// TwinCAT 3 PLC project motor_test1
// ProgramVersion: 3.1.0.9
// libraries:
//   VisuElem3DPath, 3.5.4.0 (System)
//   VisuElemMeter, 3.5.4.0 (System)
//   VisuElems, 3.5.4.10 (System)
//   VisuElemsSpecialControls, 3.5.4.10 (System)
//   VisuElemsWinControls, 3.5.4.10 (System)
//   VisuElemTextEditor, 3.5.4.0 (System)
//   visuinputs, 3.5.4.0 (system)
//   VisuNativeControl, 3.5.4.0 (System)
//   Tc2_Standard, * (Beckhoff Automation GmbH)
//   Tc2_System, * (Beckhoff Automation GmbH)
//   Tc2_Utilities, * (Beckhoff Automation GmbH)
//   Tc3_Interfaces, * (Beckhoff Automation GmbH)
//   Tc3_Module, * (Beckhoff Automation GmbH)
//   VisuDialogs, * (System)
//   Tc2_MC2,3.3.8.0,Beckhoff Automation GmbH
//   Tc2_SerialCom,3.3.3.0,Beckhoff Automation GmbH
// project tree:
//   / FastTask.TcTTO, GlobalTextList.TcGTLO, PlcTask.TcTTO, Visualization Manager.TcVMO (not stored)
//   GVLs/ GVL.TcGVL
//   POUs/ allgemein.TcPOU, Background.TcPOU, BackgroundEL.TcPOU, MAIN.TcPOU, resetErrorHandling.TcPOU, SerialCom.TcPOU, visu.TcPOU, writeInArray.TcPOU (not stored)
//   VISUs/ ImageCollection.TcIPO (not stored), AutomaticMode.TcVIS, startView.TcVIS
// real-time tasks:
//   TASK PlcTask: cycle T#5ms, priority 20, ADS port 351
//   TASK FastTask: cycle T#1ms, priority 10, ADS port 350
// motion (NC):
//   TASK NC-Task 1 SAF: cycle T#2ms, priority 4, ADS port 501
//   TASK NC-Task 1 SVB: cycle T#10ms, priority 8, ADS port 511
//   AXIS Axis Y (id 1)
//     Dynamic: Acceleration=3000, Deceleration=3000, Jerk=500
//     Velo: RefSearch=10, RefSync=10, SlowManual=10, FastManual=100, Maximum=400
//     OtherSettings: AllowMotionCmdToSlave=true
//     encoder EncType=4
//       EncPara: ScaleFactorNumerator=0.015707963, Inverse=true, MaxCount=#x0000ffff
//         Inc: RefSearchInverse=true, RefSyncInverse=false
//     drive DrvType=24
//       Analog: VeloReferenz=628
//       TimeComp: TaskDelayCycles=1
//     controller CtrType=1
//       CtrPara: PriorControlFactor=1
//         PID: PosKp=10
//         Observer: BandWidth=20
//   AXIS Axis X (id 2)
//     Dynamic: Acceleration=3000, Deceleration=3000, Jerk=500
//     Velo: RefSearch=10, RefSync=10, SlowManual=10, FastManual=100, Maximum=400
//     OtherSettings: AllowMotionCmdToSlave=true
//     encoder EncType=4
//       EncPara: ScaleFactorNumerator=0.015707963, Inverse=true, MaxCount=#x0000ffff
//         Inc: RefSearchInverse=true, RefSyncInverse=false
//     drive DrvType=24
//       Analog: VeloReferenz=628
//       TimeComp: TaskDelayCycles=1
//     controller CtrType=1
//       CtrPara: PriorControlFactor=1
//         PID: PosKp=10
//         Observer: BandWidth=20
// I/O:
//   DEVICE Device 3 (EtherCAT), AmsNetId 10.15.32.48.4.1
//     Term 1 (CX1100-0004) [CX1100-0004 EtherCAT Power supply (2A E-Bus)]
//       Term 2 (EL1859) [EL1859 8Ch. Dig. Input 24V, 3ms, 8Ch. Dig. Output 24V, 0.5A]
//       Term 3 (EL6001) [EL6001 Interface (RS232)]
//       Term 4 (EL7041) [EL7041 1Ch. Stepper motor output stage (50V, 5A)]
//       Term 5 (EL7041) [EL7041 1Ch. Stepper motor output stage (50V, 5A)]
//       Term 6 (EL9011) [EL9011 End Terminal]
// variable links:
//   NC-Task 1 SAF/Axes/Axis X <-> Device 3 (EtherCAT)/Term 1 (CX1100-0004)/Term 5 (EL7041)
//     Drive/Inputs/In/nState1 @bit 3 <-> STM Status/Status/Error
//     Drive/Inputs/In/nState1 @bit 5 <-> STM Status/Status/Moving negative
//     Drive/Inputs/In/nState1 @bit 4 <-> STM Status/Status/Moving positive
//     Drive/Inputs/In/nState1 @bit 1 <-> STM Status/Status/Ready
//     Drive/Inputs/In/nState1 <-> STM Status/Status/Ready to enable
//     Drive/Inputs/In/nState1 @bit 6 <-> STM Status/Status/Torque reduced
//     Drive/Inputs/In/nState1 @bit 2 <-> STM Status/Status/Warning
//     Drive/Inputs/In/nState2 @bit 4 <-> STM Status/Status/Digital input 2
//     Drive/Inputs/In/nState2 @bit 5 <-> STM Status/Status/Sync error
//     Drive/Inputs/In/nState2 @bit 7 <-> STM Status/Status/TxPDO Toggle
//     Drive/Inputs/In/nState4 @bit 1 <-> WcState/InputToggle
//     Drive/Inputs/In/nState4 <-> WcState/WcState
//     Drive/Outputs/Out/nCtrl1 <-> STM Control/Control/Enable
//     Drive/Outputs/Out/nCtrl1 @bit 2 <-> STM Control/Control/Reduce torque
//     Drive/Outputs/Out/nCtrl1 @bit 1 <-> STM Control/Control/Reset
//     Drive/Outputs/Out/nDataOut2[0] <-> STM Velocity/Velocity
//     Enc/Inputs/In/nDataIn1[0] <-> ENC Status compact/Counter value
//     Enc/Inputs/In/nDataIn2[0] <-> ENC Status compact/Latch value
//     Enc/Inputs/In/nState1 @bit 4 <-> ENC Status compact/Status/Counter overflow
//     Enc/Inputs/In/nState1 @bit 3 <-> ENC Status compact/Status/Counter underflow
//     Enc/Inputs/In/nState1 @bit 7 <-> ENC Status compact/Status/Extrapolation stall
//     Enc/Inputs/In/nState1 <-> ENC Status compact/Status/Latch C valid
//     Enc/Inputs/In/nState1 @bit 1 <-> ENC Status compact/Status/Latch extern valid
//     Enc/Inputs/In/nState1 @bit 2 <-> ENC Status compact/Status/Set counter done
//     Enc/Inputs/In/nState2 @bit 4 <-> ENC Status compact/Status/Status of extern latch
//     Enc/Inputs/In/nState2 <-> ENC Status compact/Status/Status of input A
//     Enc/Inputs/In/nState2 @bit 1 <-> ENC Status compact/Status/Status of input B
//     Enc/Inputs/In/nState2 @bit 2 <-> ENC Status compact/Status/Status of input C
//     Enc/Inputs/In/nState2 @bit 5 <-> ENC Status compact/Status/Sync error
//     Enc/Inputs/In/nState2 @bit 7 <-> ENC Status compact/Status/TxPDO Toggle
//     Enc/Inputs/In/nState4 @bit 1 <-> WcState/InputToggle
//     Enc/Inputs/In/nState4 <-> WcState/WcState
//     Enc/Outputs/Out/nCtrl1 <-> ENC Control compact/Control/Enable latch C
//     Enc/Outputs/Out/nCtrl1 @bit 3 <-> ENC Control compact/Control/Enable latch extern on negative edge
//     Enc/Outputs/Out/nCtrl1 @bit 1 <-> ENC Control compact/Control/Enable latch extern on positive edge
//     Enc/Outputs/Out/nCtrl1 @bit 2 <-> ENC Control compact/Control/Set counter
//     Enc/Outputs/Out/nDataOut1[0] <-> ENC Control compact/Set counter value
//   NC-Task 1 SAF/Axes/Axis Y <-> Device 3 (EtherCAT)/Term 1 (CX1100-0004)/Term 4 (EL7041)
//     Drive/Inputs/In/nState1 @bit 3 <-> STM Status/Status/Error
//     Drive/Inputs/In/nState1 @bit 5 <-> STM Status/Status/Moving negative
//     Drive/Inputs/In/nState1 @bit 4 <-> STM Status/Status/Moving positive
//     Drive/Inputs/In/nState1 @bit 1 <-> STM Status/Status/Ready
//     Drive/Inputs/In/nState1 <-> STM Status/Status/Ready to enable
//     Drive/Inputs/In/nState1 @bit 6 <-> STM Status/Status/Torque reduced
//     Drive/Inputs/In/nState1 @bit 2 <-> STM Status/Status/Warning
//     Drive/Inputs/In/nState2 @bit 4 <-> STM Status/Status/Digital input 2
//     Drive/Inputs/In/nState2 @bit 5 <-> STM Status/Status/Sync error
//     Drive/Inputs/In/nState2 @bit 7 <-> STM Status/Status/TxPDO Toggle
//     Drive/Inputs/In/nState4 @bit 1 <-> WcState/InputToggle
//     Drive/Inputs/In/nState4 <-> WcState/WcState
//     Drive/Outputs/Out/nCtrl1 <-> STM Control/Control/Enable
//     Drive/Outputs/Out/nCtrl1 @bit 2 <-> STM Control/Control/Reduce torque
//     Drive/Outputs/Out/nCtrl1 @bit 1 <-> STM Control/Control/Reset
//     Drive/Outputs/Out/nDataOut2[0] <-> STM Velocity/Velocity
//     Enc/Inputs/In/nDataIn1[0] <-> ENC Status compact/Counter value
//     Enc/Inputs/In/nDataIn2[0] <-> ENC Status compact/Latch value
//     Enc/Inputs/In/nState1 @bit 4 <-> ENC Status compact/Status/Counter overflow
//     Enc/Inputs/In/nState1 @bit 3 <-> ENC Status compact/Status/Counter underflow
//     Enc/Inputs/In/nState1 @bit 7 <-> ENC Status compact/Status/Extrapolation stall
//     Enc/Inputs/In/nState1 <-> ENC Status compact/Status/Latch C valid
//     Enc/Inputs/In/nState1 @bit 1 <-> ENC Status compact/Status/Latch extern valid
//     Enc/Inputs/In/nState1 @bit 2 <-> ENC Status compact/Status/Set counter done
//     Enc/Inputs/In/nState2 @bit 4 <-> ENC Status compact/Status/Status of extern latch
//     Enc/Inputs/In/nState2 <-> ENC Status compact/Status/Status of input A
//     Enc/Inputs/In/nState2 @bit 1 <-> ENC Status compact/Status/Status of input B
//     Enc/Inputs/In/nState2 @bit 2 <-> ENC Status compact/Status/Status of input C
//     Enc/Inputs/In/nState2 @bit 5 <-> ENC Status compact/Status/Sync error
//     Enc/Inputs/In/nState2 @bit 7 <-> ENC Status compact/Status/TxPDO Toggle
//     Enc/Inputs/In/nState4 @bit 1 <-> WcState/InputToggle
//     Enc/Inputs/In/nState4 <-> WcState/WcState
//     Enc/Outputs/Out/nCtrl1 <-> ENC Control compact/Control/Enable latch C
//     Enc/Outputs/Out/nCtrl1 @bit 3 <-> ENC Control compact/Control/Enable latch extern on negative edge
//     Enc/Outputs/Out/nCtrl1 @bit 1 <-> ENC Control compact/Control/Enable latch extern on positive edge
//     Enc/Outputs/Out/nCtrl1 @bit 2 <-> ENC Control compact/Control/Set counter
//     Enc/Outputs/Out/nDataOut1[0] <-> ENC Control compact/Set counter value
//   motor_test1/motor_test1 Instance <-> Device 3 (EtherCAT)/Term 1 (CX1100-0004)/Term 2 (EL1859)
//     PlcTask Inputs/GVL.bEmergencyPressed <-> Channel 1/Input
//   motor_test1/motor_test1 Instance <-> Device 3 (EtherCAT)/Term 1 (CX1100-0004)/Term 3 (EL6001)
//     FastTask Inputs/BackgroundEL.stIn_EL6001 @bit {16..184 step 8} <-> COM Inputs/Data In {0..21}  (22 links)
//     FastTask Inputs/BackgroundEL.stIn_EL6001 <-> COM Inputs/Status
//     FastTask Outputs/BackgroundEL.stOut_EL6001 <-> COM Outputs/Ctrl
//     FastTask Outputs/BackgroundEL.stOut_EL6001 @bit {16..184 step 8} <-> COM Outputs/Data Out {0..21}  (22 links)
//   motor_test1/motor_test1 Instance <-> Device 3 (EtherCAT)/Term 1 (CX1100-0004)/Term 4 (EL7041)
//     PlcTask Inputs/MAIN.diY <-> STM Status/Status/Digital input 1
//   motor_test1/motor_test1 Instance <-> Device 3 (EtherCAT)/Term 1 (CX1100-0004)/Term 5 (EL7041)
//     PlcTask Inputs/MAIN.diX <-> STM Status/Status/Digital input 1
//   motor_test1/motor_test1 Instance <-> NC-Task 1 SAF/Axes/Axis X
//     PlcTask Inputs/GVL.axisX.NcToPlc <-> Outputs/ToPlc
//     PlcTask Outputs/GVL.axisX.PlcToNc <-> Inputs/FromPlc
//   motor_test1/motor_test1 Instance <-> NC-Task 1 SAF/Axes/Axis Y
//     PlcTask Inputs/GVL.axisY.NcToPlc <-> Outputs/ToPlc
//     PlcTask Outputs/GVL.axisY.PlcToNc <-> Inputs/FromPlc

CONFIGURATION motor_test1
    RESOURCE PLC ON TwinCAT3
        TASK FastTask(INTERVAL := T#1ms, PRIORITY := 10);
        TASK PlcTask(INTERVAL := T#5ms, PRIORITY := 20);
        PROGRAM Background WITH FastTask : Background;
        PROGRAM MAIN WITH PlcTask : MAIN;
    END_RESOURCE
END_CONFIGURATION

// ---- GVLs/GVL.TcGVL
VAR_GLOBAL
	BuffTX: ComBuffer;
	BuffRX: ComBuffer;
	acutalForceValue: INT;
	globalForceValueArrived: BOOL;
	respondOfORder: STRING;
	(*errors*)
	globalErrorDetect: BOOL :=FALSE;
	globalErrorFromUC:STRING;
	posAxisZ: INT;
	respondI : SR;
	respondD : SR;
	respondH : SR;
	respondP : SR;
	respondOK : SR;
	respondStartetUp : SR;
	emergencyStopToMuchForce : SR;
	errorNoSignalFromUc : SR;
	motorXYNoPower : SR;
	unequalLoadThanExpected : SR;
	zAxisNotMoving : SR;
	cycleFinished : BOOL;
	counterSerialCom : UDINT;
	(*values for visu*)
	maxForceValuePos : INT;
	maxForceValueNeg : INT;
	(*Function declaration for the stepper Motor control*)
	axisX, axisY : AXIS_REF;
	powerX, powerY : MC_Power;
	resetX, resetY : MC_Reset;
	homeX, homeY : MC_Home;
	moveAbsX, moveAbsY, moveAbsNewY : MC_MoveAbsolute;
	buffermoveAbsY: MC_BufferMode := MC_Aborting;
	posAxisX, posAxisY: MC_ReadActualPosition;
	SCL : SerialCom;
	(* read status of the motors x and y *)
	readInfoAxisX, readInfoAxisY : MC_ReadStatus;
	(*for the VISU*)
	realVisuPosX: REAL;
	realVisuPosY: REAL;
	intVisuPosZ: INT;
	realVisuDiskX: REAL;
	realVisuDiskY: REAL;
	(* state of the programm *)
	iState: INT; //statemachine from the Programm
	(* boolsche variablen *)
	bLoaded: BOOL := FALSE;
	bEnable : BOOL := FALSE;
	bReset : BOOL := FALSE;	
	bEmergencyPressed AT %I* : BOOL;
	bStartViewPressed : BOOL := FALSE;
	(* errer variables*)
	errorOccurd : BOOL;
	(* other functiosn *)
	waitWithEnable: TOF; //TOF  after emergency was reseted
	noSiganlFromU: TOF; //TOF  after emergency was reseted
	rTrigStartCycle:r_trig;
	rTrigStartViewPressed:r_trig;
	fTrigReset: f_trig;
	waitToLongForRespond : TON;
	setError : SR;
	NotHomed :SR;
	(*Positions from the Manipulator*)
	posHomeVelocityX: LREAL := 50.0;
	posHomeVelocityY: LREAL := 50.0;
	posRepositoryVelocityX: LREAL :=50.0;
	posRepositoryVelocityY: LREAL := 50.0;
	posPrepositioningVelocityX: LREAL := 50.0;
	posPrepositioningVelocityY: LREAL := 50.0;
	(*Positions from the Manipulator*)
	posHomeX: LREAL := 15.0;
	posHomeY: LREAL := 400.0;
	posRepositoryX: LREAL :=134.5;
	posRepositoryY: LREAL := 0.2;
	posPrepositioningX: LREAL := posRepositoryX;
	posPrepositioningY: LREAL := 125;
END_VAR

// ---- POUs/Background.TcPOU
PROGRAM Background

(*
The SerialLineControl function block is supposed to be called in every PLC cycle.
It communicates with the serial line hardware device and transmits or receives data.
The SerialLineControl can be called in the standard task (e.g.for PcCOM port usage) 
or in a separate fast task (e.g.for terminal usage) as well.
A fast separate task will be necessary at high baud rates or with KL6001 terminals 
which have a small process image (3 or 5 data bytes only)
*)

(* background communication with the EL6001 terminal *)
BackgroundEL();

END_PROGRAM

// ---- POUs/BackgroundEL.TcPOU
PROGRAM BackgroundEL
VAR
	/// background communication with the EL6001 terminal 
	fbEL6001Ctrl: SerialLineControl;
	bEL6001CtrlError: BOOL;
	eEL6001CtrlErrorID: ComError_t;
	/// linked to the EL6001 in the TwinCAT System Manager 
	stIn_EL6001 AT %I*: EL6inData22B;
	/// linked to the EL6001 in the TwinCAT System Manager 
	stOut_EL6001 AT %Q*: EL6outData22B;
END_VAR

(*
The SerialLineControl function block is supposed to be called in every PLC cycle.
It communicates with the serial line hardware device and transmits or receives data.
The SerialLineControl can be called in the standard task (e.g.for PcCOM port usage) 
or in a separate fast task (e.g.for terminal usage) as well.
A fast separate task will be necessary at high baud rates or with KL6001 terminals 
which have a small process image (3 or 5 data bytes only)
*)

(* background communication with the EL6001 terminal *)
fbEL6001Ctrl(
	Mode:= SERIALLINEMODE_EL6_22B, 
	pComIn:= ADR(stIn_EL6001), 
	pComOut:= ADR(stOut_EL6001), 
	SizeComIn:= SIZEOF(stIn_EL6001), 
	Error=> , 
	ErrorID=> , 
	TxBuffer:= BuffTX, 
	RxBuffer:= BuffRX );
IF fbEL6001Ctrl.Error THEN
	bEL6001CtrlError := TRUE;
	eEL6001CtrlErrorID := fbEL6001Ctrl.ErrorID;
END_IF

END_PROGRAM

// ---- POUs/MAIN.TcPOU
PROGRAM MAIN
VAR CONSTANT 
	BufStart:INT:=  1;      // Start-Index
 	BufEnd:INT:=  100;   // End-Index
END_VAR

VAR
	diX, diY AT %I* : BOOL;
	(*boole variables*)
	bStart :BOOL := FALSE;
	bMoveHome : BOOL := FALSE;
	bDauerlauf : BOOL := FALSE;
	i: INT;
	btest : BOOL;
		btestZwei : bool;
	btesDrei: BOOL;
END_VAR

allgemein();

posAxisX(Axis:= axisX, Enable:= TRUE , Valid=> , Busy=> , Error=> , ErrorID=> , Position=> );
posAxisY(Axis:= axisY, Enable:= TRUE, Valid=> , Busy=> , Error=> , ErrorID=> , Position=> );

powerX(Axis:= axisX, Enable:= bEnable, Enable_Positive:= bEnable, Enable_Negative:= bEnable, Override:= 100, BufferMode:= , Options:= , Status=> , Busy=> , Active=> , Error=> , ErrorID=> );
powerY(Axis:= axisY, Enable:= bEnable, Enable_Positive:= bEnable, Enable_Negative:= bEnable, Override:= 100, BufferMode:= , Options:= , Status=> , Busy=> , Active=> , Error=> , ErrorID=> );

resetX(Axis:= axisX, Execute:= , Done=> , Busy=> , Error=> , ErrorID=> );
resetY(Axis:= axisY, Execute:= , Done=> , Busy=> , Error=> , ErrorID=> );

homeX(Axis:= axisX, Execute:= , Position:= 0 , HomingMode:= , BufferMode:= , Options:= , bCalibrationCam:= NOT diX, Done=> , Busy=> , Active=> , CommandAborted=> , Error=> , ErrorID=> );
homeY(Axis:= axisY, Execute:= , Position:= 0 , HomingMode:= , BufferMode:= , Options:= , bCalibrationCam:= NOT diY, Done=> , Busy=> , Active=> , CommandAborted=> , Error=> , ErrorID=> );	

moveAbsX(Axis:= axisX, Execute:= , Position:= , Velocity:= , Acceleration:= , Deceleration:= , Jerk:= , BufferMode:= , Options:= , Done=> , Busy=> , Active=> , CommandAborted=> , Error=> , ErrorID=> );

moveAbsY(Axis:= axisY, Execute:= , Position:= , Velocity:= , Acceleration:= , Deceleration:= , Jerk:= , BufferMode:= buffermoveAbsY, Options:= , Done=> , Busy=> , Active=> , CommandAborted=> , Error=> , ErrorID=> );

moveAbsNewY(Axis:= axisY, Execute:= , Position:= , Velocity:= , Acceleration:= , Deceleration:= , Jerk:= , BufferMode:= buffermoveAbsY, Options:= , Done=> , Busy=> , Active=> , CommandAborted=> , Error=> , ErrorID=> );	

SCL(Crtl:= , bSend:= , ReceivedString=> , bNewString=> , bSendBusy=> , bStringReceived=> );
	
	rTrigStartCycle(CLK:= bStart , Q=> );
	CASE iState OF
		
	0:	IF (*rTrig.Q AND *)powerX.Status AND powerY.Status THEN
			iState := iState + 1;
		END_IF

	1:	SCL.Crtl := 'I';
		SCL.bSend := TRUE;
		respondOfORder := '';
		istate := 2;

	2:	IF NOT SCL.bSendBusy THEN
			SCL.bSend := FALSE;
			istate := 3;
		END_IF

	3:	IF waitToLongForRespond.Q THEN
			istate := 1;
		END_IF
		IF respondI.Q1 THEN
			respondI.RESET := TRUE;
			respondI.SET1 := FALSE;
			istate := 5;
		END_IF	
	
	5:		resetX.Execute :=TRUE;
			resetY.Execute :=TRUE;
			iState := 10;
		
	10:	IF resetX.Done AND resetY.Done THEN
			resetX.Execute := FALSE;
			resetY.Execute := FALSE;
			iState :=  iState + 5;
		END_IF
		
	15: IF NOT readInfoAxisX.Status.Homed or NOT readInfoAxisY.Status.Homed THEN
		homeX.Execute := TRUE;
		homeY.Execute := TRUE;
		iState := 20;
		ELSE
			iState := 21; //--> if already referenced, go home position
		END_IF
	20:	IF homeX.Done AND homeY.Done THEN
			homeX.Execute := FALSE;
			homeY.Execute := FALSE;
			NotHomed.RESET := FALSE;
			iState := 21;		
		END_IF
	21:			moveAbsY.Velocity := posHomeVelocityY;
				moveAbsY.Position := posHomeY;
				moveAbsY.Execute := TRUE;

			IF posAxisY.Position > posPrepositioningY THEN
				moveAbsX.Velocity := posHomeVelocityX;
				moveAbsX.Position := posHomeX;
				moveAbsX.Execute := TRUE;
				iState :=  25;
			END_IF

	25:	IF 	moveAbsX.Done AND moveAbsY.Done THEN
			moveAbsX.Execute:= FALSE;
			moveAbsY.Execute:= FALSE;
			respondH.RESET := TRUE;
			respondH.SET1 := FALSE;
			iState :=  26;
		END_IF
		
	(*this starts a new cycle, depending on the load*)
	26:	IF rTrigStartCycle.Q OR bDauerlauf THEN
			IF bLoaded THEN
				iState :=  125;
			ELSE
				iState :=  27;
			END_IF
			respondD.RESET := TRUE;
			respondD.SET1 := FALSE;
			respondH.RESET := TRUE;
			respondH.SET1 := FALSE;
			respondP.RESET := TRUE;
			respondP.SET1 := FALSE;
			cycleFinished := FALSE;
		END_IF				
		
	27:		moveAbsX.Velocity := posRepositoryVelocityX;
			moveAbsX.Position := posRepositoryX;
			moveAbsX.Execute := TRUE;
			moveAbsY.Velocity := posRepositoryVelocityY;
			moveAbsY.Position :=posRepositoryY;
			moveAbsY.Execute := TRUE;
			iState :=  28;
			maxForceValuePos := 0;
			maxForceValueNeg := 0;

	28: 	SCL.Crtl := 'P'; // vorpositionieren
			SCL.bSend := TRUE;
			iState :=  29;
		
	29:	IF NOT SCL.bSendBusy THEN
			SCL.bSend := FALSE;
			SCL.Crtl := '';
			istate := 30;
		END_IF
		
	30:	IF waitToLongForRespond.Q THEN
			istate := 28;
			END_IF
		IF 	moveAbsX.Done AND moveAbsY.Done AND respondP.Q1 THEN
			moveAbsX.Execute:= FALSE;
			moveAbsY.Execute:= FALSE;
			respondP.RESET := TRUE;
			respondP.SET1 := FALSE;
			iState := 31;
		END_IF
		
	31:	SCL.Crtl := 'D';
		SCL.bSend := TRUE;
		istate := 32;
		
	32:	IF NOT SCL.bSendBusy THEN
			SCL.bSend := FALSE;
			SCL.Crtl := '';
			istate := 33;
		END_IF

	33:	IF waitToLongForRespond.Q THEN
			istate := 31;
			END_IF
		IF respondD.Q1 THEN //Move Down
			respondD.RESET := TRUE;
			respondD.SET1 := FALSE;
			bLoaded := TRUE;
			cycleFinished :=TRUE;
			istate := 35;
		END_IF	
		
	35:		IF NOT respondD.Q1 THEN
				moveAbsY.Velocity := posHomeVelocityY;
				moveAbsY.Position :=posHomeY;
				moveAbsY.Execute := TRUE;
			IF posAxisY.Position > posPrepositioningY THEN //über dem weg drausen, dan darf er fahren
				moveAbsX.Velocity := posHomeVelocityX;
				moveAbsX.Position := posHomeX;
				moveAbsX.Execute := TRUE;
				iState :=  40;
			END_IF
		
		END_IF
	40:	IF 	moveAbsX.Done AND moveAbsY.Done THEN
			moveAbsX.Execute:= FALSE;
			moveAbsY.Execute:= FALSE;
			iState := 26;
		END_IF
		
	125:	moveAbsX.Velocity := posPrepositioningVelocityX;
			moveAbsX.Position := posPrepositioningX;
			moveAbsX.Execute := TRUE;
			moveAbsY.Velocity := posPrepositioningVelocityY;
			moveAbsY.Position :=posPrepositioningY;
			moveAbsY.Execute := TRUE;
			iState :=  130;
			maxForceValuePos := 0;
			maxForceValueNeg := 0;
			
	130:	IF moveAbsX.Done THEN
				moveAbsNewY.Execute:= TRUE;
				moveAbsNewY.Velocity := posRepositoryVelocityY;
				moveAbsNewY.Position := posRepositoryY;
				moveAbsY.Execute:= FALSE;
				moveAbsX.Execute:= FALSE;
			END_IF
			IF moveAbsNewY.Done THEN
				iState := 140;
		END_IF
		
	(*135:	moveAbsX.Velocity := 	posRepositoryVelocityX;
			moveAbsX.Position := 	posRepositoryX;
			moveAbsX.Execute := 	TRUE;
			moveAbsY.Velocity :=	posRepositoryVelocityY;
			moveAbsY.Position :=	posRepositoryY;
			moveAbsY.Execute := TRUE;
			iState :=  140;*)
			
	140:	IF 	(*moveAbsX.Done AND*) moveAbsNewY.Done THEN
			moveAbsNewY.Execute:= FALSE;
			iState :=  141;
			END_IF
			
	141:	SCL.Crtl := 'P'; //Move Up
			SCL.bSend := TRUE;
			istate := 142;
			
	142:	IF NOT SCL.bSendBusy THEN
			SCL.bSend := FALSE;
			SCL.Crtl := '';
			istate := 143;
		END_IF

	143:	IF waitToLongForRespond.Q THEN
				istate := 141;
			END_IF
			IF respondP.Q1 THEN
				respondP.RESET := TRUE;
				respondP.SET1 := FALSE;
				bLoaded := FALSE;
				cycleFinished :=TRUE;
				iState := 145;
			END_IF	
			
	145:	SCL.Crtl := 'H'; // Home pos anfahren
			SCL.bSend := TRUE;
			iState :=  150;
		
	150:	IF NOT SCL.bSendBusy THEN
				SCL.bSend := FALSE;
				SCL.Crtl := '';
				istate := 155;
			END_IF

 	155:	moveAbsY.Velocity := posHomeVelocityY;
				moveAbsY.Position := posHomeY;
				moveAbsY.Execute := TRUE;

			IF posAxisY.Position > posPrepositioningY THEN
				moveAbsX.Velocity := posHomeVelocityX;
				moveAbsX.Position := posHomeX;
				moveAbsX.Execute := TRUE;
				iState :=  160;
			END_IF
		
	160:	IF waitToLongForRespond.Q THEN
				istate := 145;
			END_IF
			IF 	moveAbsX.Done AND moveAbsY.Done AND respondH.Q1 THEN
			moveAbsX.Execute:= FALSE;
			moveAbsY.Execute:= FALSE;
			respondH.RESET := TRUE;
			respondH.SET1 := FALSE;
			iState :=  26;
		END_IF
		
	END_CASE
	
	resetErrorHandling();
	visu();

END_PROGRAM

// ---- POUs/allgemein.TcPOU
PROGRAM allgemein
VAR
END_VAR

(*safe the min and max value of the force*)
IF maxForceValuePos < acutalForceValue THEN
	maxForceValuePos := acutalForceValue;
END_IF
IF maxForceValueNeg > acutalForceValue THEN
	maxForceValueNeg := acutalForceValue;
END_IF

END_PROGRAM

// ---- POUs/resetErrorHandling.TcPOU
PROGRAM resetErrorHandling
VAR
	reset: INT := 0; //reset state machine
END_VAR

VAR CONSTANT 
	toMuchForcePositive : INT := 15000;
	toMuchForceNegative : INT := -15000;
END_VAR

respondD(SET1:= , RESET:= , Q1=> );
respondH(SET1:= , RESET:= , Q1=> );
respondI(SET1:= , RESET:= , Q1=> );
respondP(SET1:= , RESET:= , Q1=> );
respondOk(SET1:= , RESET:= , Q1=> );
respondStartetUp(SET1:= , RESET:= , Q1=> );
emergencyStopToMuchForce(SET1:= , RESET:= , Q1=> );
motorXYNoPower(SET1:= , RESET:= , Q1=> );
errorNoSignalFromUc(SET1:= , RESET:= , Q1=> );
unequalLoadThanExpected(SET1:= , RESET:= , Q1=> );
zAxisNotMoving(SET1:= , RESET:= , Q1=> );

rTrigStartViewPressed(CLK:= bStartViewPressed , Q=> );

IF respondI.Q1 THEN
		respondI.SET1 := FALSE;
END_IF

respondD.RESET := FALSE;
respondH.RESET := FALSE;
respondI.RESET := FALSE;
respondP.RESET := FALSE;
respondOK.RESET := FALSE;
respondStartetUp.RESET := FALSE;
emergencyStopToMuchForce.RESET := FALSE;
motorXYNoPower.RESET := FALSE;
errorNoSignalFromUc.RESET := FALSE;
unequalLoadThanExpected.RESET := FALSE;
zAxisNotMoving.RESET:=FALSE;

(*read status from x and y*)
readInfoAxisX(Axis:= axisX, Enable:= TRUE, Valid=> , Busy=> , Error=> , ErrorID=> , ErrorStop=> , Disabled=> , Stopping=> , StandStill=> , DiscreteMotion=> , ContinuousMotion=> , SynchronizedMotion=> , Homing=> , ConstantVelocity=> , Accelerating=> , Decelerating=> , Status=> );
readInfoAxisY(Axis:= axisY, Enable:= TRUE, Valid=> , Busy=> , Error=> , ErrorID=> , ErrorStop=> , Disabled=> , Stopping=> , StandStill=> , DiscreteMotion=> , ContinuousMotion=> , SynchronizedMotion=> , Homing=> , ConstantVelocity=> , Accelerating=> , Decelerating=> , Status=> );

(* wait to seconds to give the stepper motor drivers a little time to built DC link*)
waitWithEnable(IN:= bEmergencyPressed, PT:= T#2S, Q=> , ET=> );

(* if no respond from the uC in a little time, the nsend command again*)
waitToLongForRespond(IN:= 	iState = 33  OR iState = 143 OR iState =3 OR iState = 30, PT:= T#10S, Q=> , ET=> );

zAxisNotMoving.SET1:= (globalErrorFromUC = '2E');

(* Ungleich soll beladung *)
IF (iState = 26 OR iState = 0) AND ((acutalForceValue > -200 AND bLoaded) OR (acutalForceValue < -700 AND NOT bLoaded))THEN
	unequalLoadThanExpected.SET1:=TRUE;
END_IF

(* error if no respond from uC*)
errorNoSignalFromUc.SET1 := NOT noSiganlFromU.Q;

(* trigger after restart from emergency *)
fTrigReset(CLK:= waitWithEnable.Q, Q=> );

(* set if we ar not homed*)
NotHomed(SET1:= NOT readInfoAxisX.Status.Homed OR NOT readInfoAxisY.Status.Homed, RESET:= , Q1=> );
motorXYNoPower.SET1 :=  readInfoAxisY.ErrorStop OR readInfoAxisX.ErrorStop;
(* Status not ok but Emergency is ok*)
globalErrorDetect := motorXYNoPower.Q1 OR respondStartetUp.Q1 OR emergencyStopToMuchForce.Q1 OR bEmergencyPressed OR errorNoSignalFromUc.Q1 OR unequalLoadThanExpected.Q1 OR zAxisNotMoving.Q1;
(* set error *)
setError(SET1:=globalErrorDetect, RESET:= , Q1=> );

CASE reset OF
0:	IF fTrigReset.Q OR ((setError.Q1 OR NotHomed.SET1) AND (bReset OR rTrigStartViewPressed.Q)) THEN
		reset := 5;
		iState := 0;
		bEnable := FALSE;
		globalErrorDetect := FALSE;
		setError.RESET :=TRUE;
		respondStartetUp.RESET := TRUE;
		bLoaded := FALSE;
		respondStartetUp.SET1 := FALSE;
		emergencyStopToMuchForce.RESET := TRUE;
		emergencyStopToMuchForce.SET1 := FALSE;
		motorXYNoPower.SET1 := FALSE;
		motorXYNoPower.RESET := TRUE;
		errorNoSignalFromUc.SET1 := FALSE;
		errorNoSignalFromUc.RESET := TRUE;
		unequalLoadThanExpected.SET1:= FALSE;
		unequalLoadThanExpected.RESET := TRUE;
		zAxisNotMoving.SET1 := FALSE;
		zAxisNotMoving.RESET := TRUE;
		respondI.RESET := TRUE;
		respondI.SET1 := FALSE;
		respondD.RESET := TRUE;
		respondD.SET1 := FALSE;
		respondH.RESET := TRUE;
		respondH.SET1 := FALSE;
		maxForceValuePos := 0;
		maxForceValueNeg := 0;
	END_IF
5:	resetX.Execute :=TRUE;
	resetY.Execute :=TRUE;
	setError.RESET :=FALSE;
	reset := 10;
	
10:	IF resetX.Done AND resetY.Done THEN
		resetX.Execute := FALSE;
		resetY.Execute := FALSE;
		reset :=  15;
	END_IF
15: bEnable := TRUE;
	reset  := 0;
END_CASE

(* if to much force --> emergency stop!*)
IF (acutalForceValue > toMuchForcePositive) OR (acutalForceValue < toMuchForceNegative) THEN
	emergencyStopToMuchForce.SET1 := TRUE;
END_IF



(*reset all movements and sending*)
IF setError.Q1 THEN
	iState := 0;
	homeX.Execute := FALSE;
	homeY.Execute := FALSE;
	moveAbsX.Execute:= FALSE;
	moveAbsY.Execute:= FALSE;
	moveAbsNewY.Execute:= FALSE;
	bEnable := FALSE;
	SCL.bSend := FALSE;
	SCL.Crtl := '';
END_IF

END_PROGRAM

// ---- POUs/visu.TcPOU
PROGRAM visu
VAR
	//stringErrorText : WSTRING; //error texts for visu
	//stringMessageText : WSTRING;
	//stringDebugText : WSTRING;
	stringErrorText: ARRAY [1..20] OF STRING;
	stringMessageText: ARRAY [1..20] OF STRING;
	stringDebugText: ARRAY [1..20] OF STRING;
	forceMemoryDrop: writeInArray;
	forceMemoryPick: writeInArray;
	zaehl: INT := 1;
	getTime: GETSYSTEMTIME;
	
	ActSystemTime1: T_ULARGE_INTEGER ;
    ActSystemTime2: T_ULARGE_INTEGER ;
    UInt64TimeDif: T_ULARGE_INTEGER ;
    TimeDifSec: LREAL;
    bZeitmess: BOOL;
    fStartflanke: R_TRIG;
    fStopflanke: F_TRIG;
END_VAR

forceMemoryDrop(i_iState:= iState, i_actualForceValue:= acutalForceValue, i_bLoaded:= TRUE, io_ValueArrived:= globalForceValueArrived);
forceMemoryPick(i_iState:= iState, i_actualForceValue:= acutalForceValue, i_bLoaded:= FALSE, io_ValueArrived:= globalForceValueArrived);

    bZeitmess:= iState > 26;
fStartflanke(CLK:= bZeitmess);
IF fStartflanke.Q THEN
    getTime(timeLoDW=> ActSystemTime1.dwLowPart,timeHiDW=> ActSystemTime1.dwHighPart);
END_IF
fStopflanke(CLK:= bZeitmess);
IF bZeitmess THEN
    getTime(timeLoDW=> ActSystemTime2.dwLowPart, timeHiDW=> ActSystemTime2.dwHighPart);
    UInt64TimeDif:= UInt64Sub64(ActSystemTime2, ActSystemTime1);
    TimeDifSec:= UINT64_TO_LREAL(UInt64TimeDif) / LREAL#10000000;
END_IF

(* pos of x and y for the visu*)
IF readInfoAxisX.Status.Homed AND readInfoAxisY.Status.Homed	THEN
realVisuPosX := posAxisX.Position * 1.5;
realVisuPosY := (posAxisY.Position * (-1.0) + 10) *1.7;
//realVisuPosX := ABS (realVisuPosX);
ELSE
realVisuPosX := 0.0;
realVisuPosY := 0.0;	
END_IF

IF bLoaded THEN
	realVisuDiskX := realVisuPosX; (* - posRepositoryX * 1.5;*)
	realVisuDiskY := realVisuPosY; (*- (posRepositoryY * (-1.0) + 10) *2.0;	*)
ELSE
	realVisuDiskX := posRepositoryX * 1.5;
	realVisuDiskY := (posRepositoryY * (-1.0) + 10) *2.0;
END_IF

IF iState > 3 THEN
intVisuPosZ := (posAxisZ) *2;
ELSE
intVisuPosZ := 0;	
END_IF

(*prepare cycle finished*)

(* visu texts *)

MEMSET(ADR(stringErrorText), 0, SIZEOF(stringErrorText));
MEMSET(ADR(stringMessageText), 0, SIZEOF(stringMessageText));
MEMSET(ADR(stringDebugText), 0, SIZEOF(stringDebugText));

zaehl := 1;
(* error messages *)
IF NOT readInfoAxisX.Status.Homed OR NOT readInfoAxisY.Status.Homed THEN
	stringErrorText[zaehl]:= CONCAT(STR1:= stringErrorText[zaehl], STR2:= 'Not referenced in X/Y');
	zaehl := zaehl + 1;
END_IF

IF  globalErrorDetect THEN
	stringErrorText[zaehl]:= CONCAT(STR1:= stringErrorText[zaehl], STR2:= 'Failure');
	zaehl := zaehl + 1;
END_IF

IF  bEmergencyPressed THEN
	stringErrorText[zaehl]:= CONCAT(STR1:= stringErrorText[zaehl], STR2:= 'Emergency Stop');
	zaehl := zaehl + 1;
END_IF

IF  emergencyStopToMuchForce.Q1 THEN
	stringErrorText[zaehl]:= CONCAT(STR1:= stringErrorText[zaehl], STR2:= 'too much Force');
	zaehl := zaehl + 1;
END_IF

IF motorXYNoPower.Q1 THEN
	stringErrorText[zaehl]:= CONCAT(STR1:= stringErrorText[zaehl], STR2:= 'Not referenced in X/Y');	
	zaehl := zaehl + 1;
END_IF

IF errorNoSignalFromUc.Q1 THEN
	stringErrorText[zaehl]:= CONCAT(STR1:= stringErrorText[zaehl], STR2:= 'error connection lost to uC');
	zaehl := zaehl + 1;
END_IF

IF unequalLoadThanExpected.Q1 THEN
	stringErrorText[zaehl]:= CONCAT(STR1:= stringErrorText[zaehl], STR2:= 'load unequal than expected');	
	zaehl := zaehl + 1;
END_IF

IF zAxisNotMoving.Q1 THEN
	stringErrorText[zaehl]:= CONCAT(STR1:= stringErrorText[zaehl], STR2:= 'z-axis Error');	
	zaehl := zaehl + 1;
END_IF

(* massage textes *)
	zaehl := 1;
IF acutalForceValue > -200  THEN
	stringMessageText[zaehl]:= CONCAT(STR1:= stringMessageText[zaehl], STR2:= 'The object is successfully dropped');
	zaehl := zaehl + 1;
END_IF

IF acutalForceValue < -700 THEN
	stringMessageText[zaehl]:= CONCAT(STR1:= stringMessageText[zaehl], STR2:= 'The object is successfully grabbed');
	zaehl := zaehl + 1;
END_IF


IF iState = 26 AND cycleFinished THEN
	stringMessageText[zaehl]:= CONCAT(STR1:= stringMessageText[zaehl], STR2:= 'Cycle successfully finished');
	zaehl := zaehl + 1;
END_IF

(* debug messages *)
	zaehl := 1;
IF bLoaded THEN	
	stringDebugText[zaehl]:= CONCAT(STR1:= stringDebugText[zaehl], STR2:= 'Load');
	zaehl := zaehl + 1;
ELSE
	stringDebugText[zaehl]:= CONCAT(STR1:= stringDebugText[zaehl], STR2:= 'No Load');
	zaehl := zaehl + 1;
END_IF

stringDebugText[zaehl]:= CONCAT(STR1:= stringDebugText[zaehl], STR2:= 'State PLC: ');
stringDebugText[zaehl]:= CONCAT(STR1:= stringDebugText[zaehl], STR2:= INT_TO_STRING (iState));
zaehl := zaehl + 1;
stringDebugText[zaehl]:= CONCAT(STR1:= stringDebugText[zaehl], STR2:= 'Error from uC:');
stringDebugText[zaehl]:= CONCAT(STR1:= stringDebugText[zaehl], STR2:= globalErrorFromUC);
zaehl := zaehl + 1;

END_PROGRAM

// ---- POUs/SerialCom.TcPOU
FUNCTION_BLOCK SerialCom
VAR_INPUT
	Crtl: STRING;
	bSend: BOOL;
END_VAR
VAR_OUTPUT
	ReceivedString: STRING;
	bNewString: BOOL;
	bSendBusy: BOOL;
	bStringReceived: BOOL;
END_VAR
(*VAR_IN_OUT
	IOrespondOfORder: STRING;
END_VAR*)
VAR
	//DataIn AT %I*: EL6inData22B;
	//DataOut AT %Q*: EL6outData22B;
	SerialLineCtrl: SerialLineControl;
	//BuffTX: ComBuffer;
	//BuffRX: ComBuffer;
	clearbuff: ClearComBuffer;
	SendString: SendString;
	RecString: ReceiveString;
	istate: INT;
	rtrig: r_trig;
	test: ReceiveByte;
	bTest: BYTE;
	bByteReceived : BOOL := FALSE;
	bBuffer: BYTE;
	arrForceValues : ARRAY [1..1000] OF INT;

	lengtOfReceivedString: INT;
	strTemp : STRING(255);
	posSuffix: INT;
	stest :STRING;
	
	posFirstSlash: INT;
	posSecondSlash: INT;
	posThirdSlash: INT;
	posHash: INT;
END_VAR

SendString(SendString:= , Busy=> , Error=> , TXbuffer:= BuffTX);
RecString(Prefix:= , Suffix:= '$N', Timeout:= T#2S, Reset:= , StringReceived=> , 	Busy=> , 	Error=> , 	RxTimeout=> , 	ReceivedString:= ReceivedString, 	RXbuffer:= BuffRX);
posHash := FIND (ReceivedString,'#');
posSuffix := FIND (ReceivedString,'$R');
posFirstSlash := FIND (ReceivedString,'/');
strTemp := MID (ReceivedString,posSuffix - posFirstSlash-1,posFirstSlash+1);
posSecondSlash := FIND (strTemp,'/') + posFirstSlash;
strTemp := MID (ReceivedString,posSuffix - posSecondSlash-1,posSecondSlash+1);
posThirdSlash := FIND (strTemp,'/') + posSecondSlash;

lengtOfReceivedString:=LEN(STR:= ReceivedString);

IF RecString.StringReceived THEN
	strTemp := MID (ReceivedString,posSecondSlash - posHash-1,posHash+1);
	acutalForceValue := STRING_TO_INT (strTemp);
	
	strTemp := MID (ReceivedString,posThirdSlash - posSecondSlash-1,posSecondSlash+1);
	posAxisZ := STRING_TO_INT (strTemp);

	globalErrorFromUC := MID (ReceivedString,posSuffix - posThirdSlash-1,posThirdSlash+1);
	
	globalForceValueArrived := TRUE;
	RecString.Reset := TRUE;

	respondOfORder := MID (ReceivedString,posFirstSlash-1,1); (* else its a respond of the Order*)
	RecString.Reset := TRUE;
	respondI.SET1 := respondOfORder = 'i';
	respondH.SET1 := respondOfORder = 'h';
	respondD.SET1 := respondOfORder = 'd';
	respondP.SET1 := respondOfORder = 'p';
	respondOK.SET1 := respondOfORder = 'ok';
	respondStartetUp.SET1 :=  respondOfORder  = 'Started up';
	respondOfORder := '';
	counterSerialCom := counterSerialCom+1;
END_IF


(* no isgnal from uC *)
noSiganlFromU(IN:= RecString.StringReceived, PT:= T#2S, Q=> , ET=> );


rtrig(CLK:= bSend, Q=> );
CASE istate OF

0:	RecString.Reset := FALSE;
	bStringReceived := FALSE;
	IF rtrig.Q THEN
		SendString.SendString := Crtl;
		bSendBusy := TRUE;
		istate := istate  + 1;
	END_IF	

1:	IF NOT SendString.Busy THEN
			SendString.SendString := '';
			(*clearbuff(Buffer:= BuffTX );*)
			istate := istate + 1;
			ReceivedString := '';
			bSendBusy := FALSE;
	END_IF

2:	IF RecString.StringReceived THEN
		bStringReceived := TRUE;
		RecString.Reset := TRUE;
		istate := 0;
	END_IF
		
END_CASE

END_FUNCTION_BLOCK

// ---- GlobalTextList.TcGTLO
TEXTLIST GlobalTextList
  41 = ' $$R $$N %s'
  42 = ' $/R $/N %s'
  46 = ' $A%s'
  40 = ' $R $N %s'
  39 = ' $R$N %s'
  45 = ' %s'
  43 = ' /R /N %s'
  44 = ' \\R \\N %s'
  47 = '"$0xA"%s'
  49 = '$#A%s'
  50 = '$0x0A%s'
  48 = '$A%s'
  5 = '%.0f'
  4 = '%.1f'
  17 = '%.2f'
  3 = '%.9f'
  16 = '%f'
  15 = '%i'
  20 = '%s'
  38 = '%s $R$N'
  33 = 'Automatic Mode'
  21 = 'continuously run'
  53 = 'Continuously Run'
  54 = 'Cylce Time [s]'
  55 = 'Cylce Time [s]:'
  13 = 'Dauverlauf'
  36 = 'Debug Messages'
  1 = 'Enable'
  14 = 'ERROR'
  37 = 'Error Messages'
  22 = 'Force / measuring points'
  23 = 'Force / measuring points Diagram'
  51 = 'Force / measuring points Diagram Drop Cycle'
  52 = 'Force / measuring points Diagram Pick Cycle'
  30 = 'Force Value in mN'
  26 = 'Force Values'
  25 = 'ForceValues'
  8 = 'Load Sim'
  31 = 'max Force Value in mN'
  24 = 'measuring points'
  32 = 'min Force Value in mN'
  2 = 'mN'
  11 = 'Position X'
  18 = 'Position X in mm'
  12 = 'Position Y'
  19 = 'Position Y in mm'
  29 = 'Position Z in mm'
  0 = 'Reference'
  7 = 'Reset'
  34 = 'Start Automatik'
  6 = 'Start Cycle'
  27 = 'Status / Error Messages'
  35 = 'Status Messages'
  9 = 'X'
  10 = 'Y'
  28 = 'Z'
END_TEXTLIST

// ---- VISUs/AutomaticMode.TcVIS
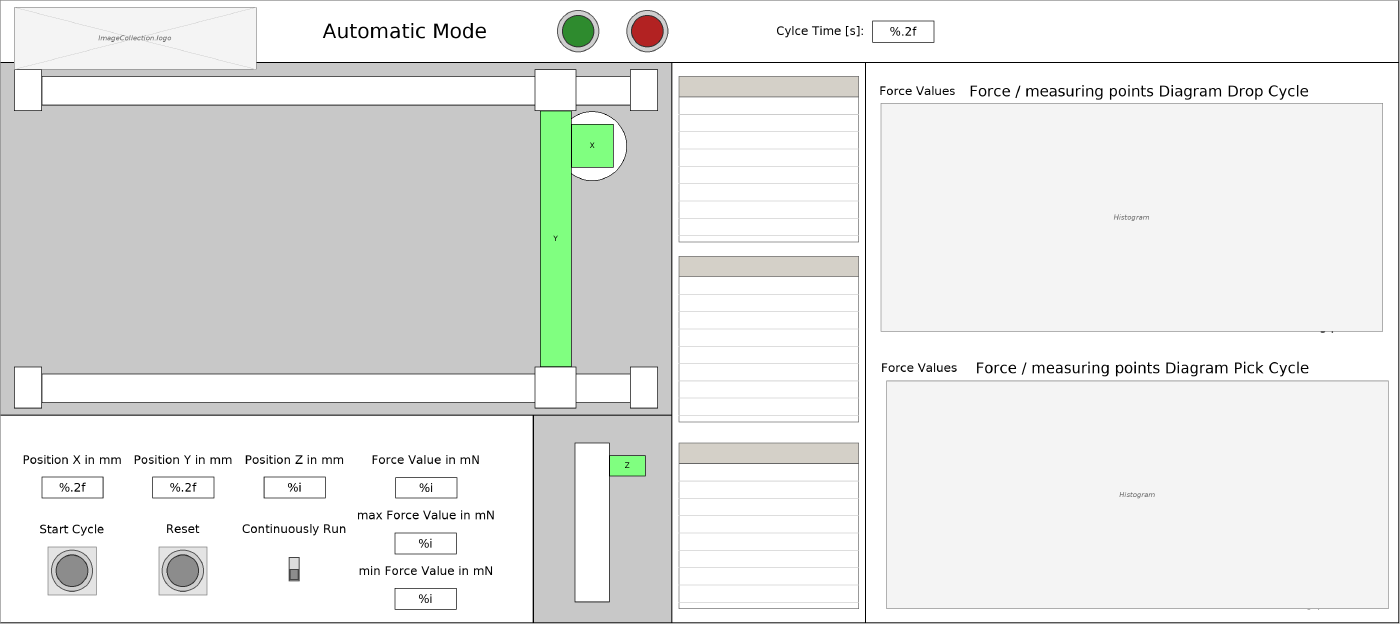
VISUALIZATION AutomaticMode  // 2022x902
    Rectangle (1250,90 770x810)
    Rectangle (0,600 770x300)
    Rectangle (970,90 280x810)
    Rectangle (0,0 2020x90)
    Rectangle (770,600 200x300)
    Rectangle (0,90 970x510)
    Ellipse (805,161 100x100)
        p3528305787: realVisuDiskY
        p2773130477: realVisuDiskX
        p874137650: realVisuDiskY
        p1126004900: realVisuDiskX
    Rectangle (60,110 852x42)
    Rectangle (60,540 852x42)
    PushSwitch (69,790 70x70), variable: MAIN.bStart, behaviour: TAP, style: Switch-PushSwitch-Gray
    Label (54,750 100x30), "Start Cycle"
    PushSwitch (229,790 70x70), variable: bReset, behaviour: TAP, style: Switch-PushSwitch-Gray
    Label (229,750 70x29), "Reset"
    Rectangle (825,179 61x63), "X", colour toggle: setError.Q1
        p3560616238: realVisuPosY
        p2738717112: realVisuPosX
    DipSwitch (390,805 70x35), variable: MAIN.bDauerlauf, behaviour: TOGGLE, style: Switch-DipSwitch-Gray
    Label (350,750 150x29), "Continuously Run"
    Rectangle (60,689 89x31), "%.2f", text variable: posAxisX.Position
    Label (30,650 149x29), "Position X in mm"
    Rectangle (220,689 89x31), "%.2f", text variable: posAxisY.Position
    Label (190,650 149x29), "Position Y in mm"
    Lamp1 (800,10 70x70), variable: NOT bEmergencyPressed AND NOT globalErrorDetect, style: Lamp-Lamp1-green
    Lamp1 (900,10 70x70), variable: bEmergencyPressed OR globalErrorDetect, style: Lamp-Lamp1-Red
    Rectangle (880,658 52x30), "Z", colour toggle: setError.Q1
        p2738717112: intVisuPosZ
    Rectangle (830,640 50x230)
    Rectangle (381,689 89x31), "%i", text variable: posAxisZ
    Label (351,650 149x29), "Position Z in mm"
    Rectangle (571,690 89x30), "%i", text variable: acutalForceValue
    Label (530,650 170x29), "Force Value in mN"
    Rectangle (570,770 89x31), "%i", text variable: maxForceValuePos
    Label (510,730 210x29), "max Force Value in mN"
    Rectangle (570,850 89x31), "%i", text variable: maxForceValueNeg
    Label (510,810 210x30), "min Force Value in mN"
    Label (460,20 250x50), "Automatic Mode"
    Group (1270,110 727x383)
        Label (120,0 510x44), "Force / measuring points Diagram Drop Cycle"
        Label (550,340 160x43), "measuring points"
        Label (0,0 110x43), "Force Values"
        Histogram (2,39 725x330), scale format: %.1f, scale -10000..3000
            p518627256: mN
            p1518820177: visu.forceMemoryDrop.sArrForceValue
            p102497268: visu.forceMemoryDrop.sArrForceValue
            p788070771: ARRAY [BufStart..BufEnd] OF INT
    Table (980,370 260x240), data array: visu.stringErrorText
        p3854506369: visu.stringErrorText[INDEX]
        p2232123230: Error Messages
    Table (980,110 260x240), data array: visu.stringMessageText
        p3854506369: visu.stringMessageText[INDEX]
        p2232123230: Status Messages
    Table (980,640 260x240), data array: visu.stringDebugText
        p3854506369: visu.stringDebugText[INDEX]
        p2232123230: Debug Messages
    Group (1270,510 735x383)
        Label (530,340 160x43), "measuring points"
        Label (120,0 520x44), "Force / measuring points Diagram Pick Cycle"
        Label (0,0 115x43), "Force Values"
        Histogram (10,40 725x330), scale format: %.1f, scale -3000..13000
            p518627256: mN
            p1518820177: visu.forceMemoryPick.sArrForceValue
            p102497268: visu.forceMemoryPick.sArrForceValue
            p788070771: ARRAY [BufStart..BufEnd] OF INT
    Rectangle (780,160 45x370), "Y", colour toggle: setError.Q1
        p3560616238: realVisuPosY
    Rectangle (772,100 60x60)
        p3560616238: realVisuPosY
    Rectangle (772,530 60x60)
        p3560616238: realVisuPosY
    Rectangle (20,100 40x60)
    Rectangle (910,100 40x60)
    Rectangle (20,530 40x60)
    Rectangle (910,530 40x60)
    Image (20,10 350x90), image: ImageCollection.logo
    Rectangle (1260,30 89x31), "%.2f", text variable: visu.TimeDifSec
    Label (1110,30 149x29), "Cylce Time [s]:"
END_VISUALIZATION

// ---- VISUs/startView.TcVIS
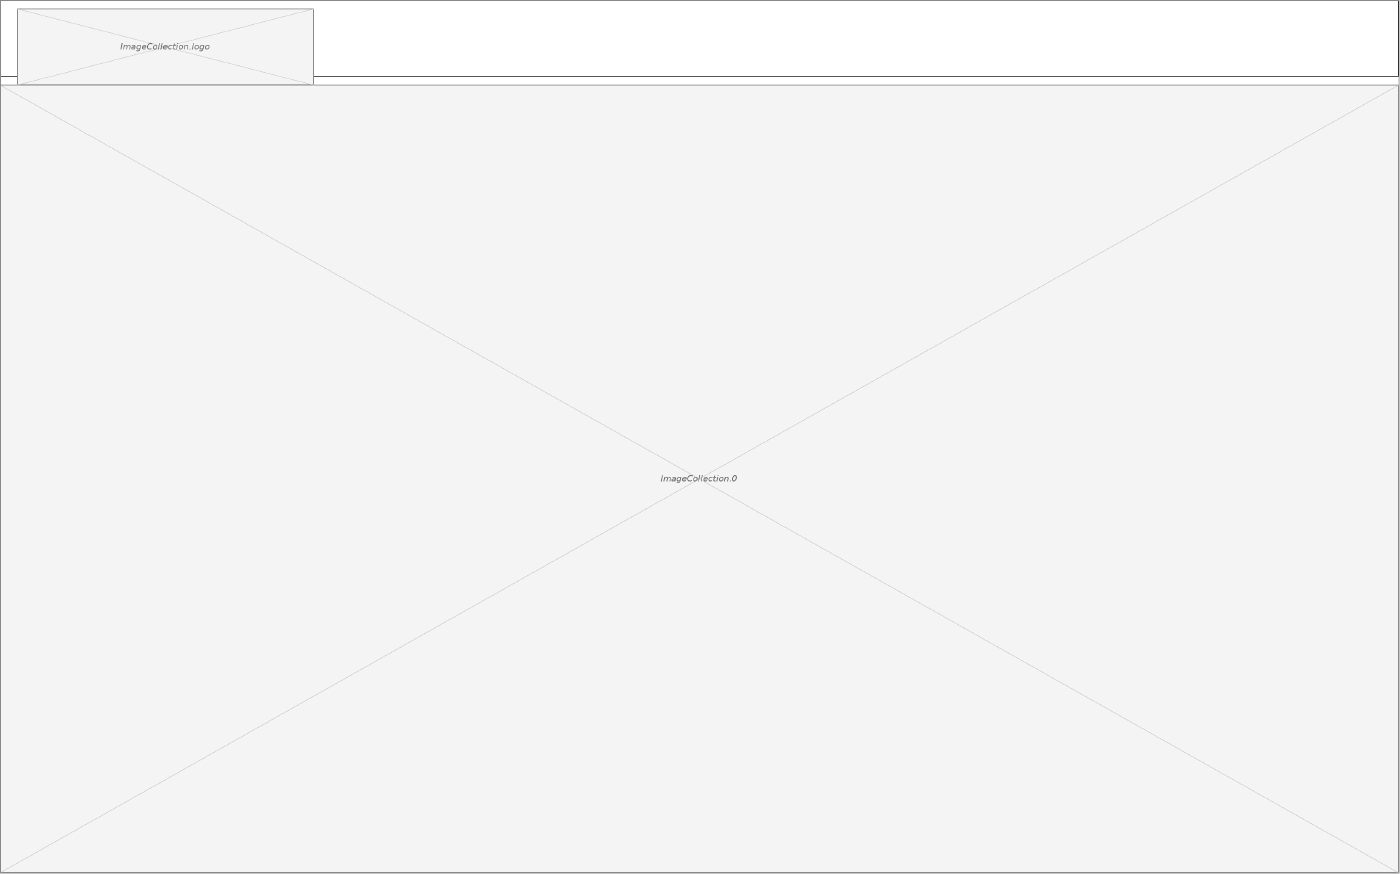
VISUALIZATION startView  // 1652x1032
    Rectangle (0,0 1650x90)
    Image (0,100 1650x930), image: ImageCollection.0
        OnMouseClick: change screen: AutomaticMode
        OnMouseClick: toggle bStartViewPressed
    Image (20,10 350x90), image: ImageCollection.logo
END_VISUALIZATION
